(* PLC project stockage, TNI-Software ControlBuild 4.00 *)
(* stored: creationDateTime 2018-09-17T17:24:47-01:00 *)

FUNCTION_BLOCK tapis_conv.stockage
  VAR_INPUT  (* CB.kind=inputVars *)
    In : BOOL := false;
    Out : BOOL := false;
  END_VAR
  VAR_OUTPUT  (* CB.kind=outputVars *)
    Nb_Pieces : INT := 0;
  END_VAR

if In = true
then 
	Nb_Pieces:=Nb_Pieces+1;
end_if;
if Out = true
then 
	Nb_Pieces:=Nb_Pieces-1;
end_if;
END_FUNCTION_BLOCK
